(* IEC 61131-3 sources: SafeDODiag/SafeDODiag (part 2) *)

(* ---- DiagAction_InterlockState.st ---- *)
ACTION DiagAction_InterlockState:

	// Check for error state transition and feedback interpretation as long as interlock-based monitoring is enabled
	IF ( Config.InterlockState.EnableMon AND ( Internal.State > SC_INIT ) AND (
		// (Choice 1) if no other monitoring is enabled
		NOT( Config.DiagCode.EnableMon OR Config.Fdbk.EnableMon OR Config.Current.EnableMon ) OR
		// (Choice 2) if DiagCode monitoring is enabled, show Interlock monitoring-based DiagText only when DiagCode indicates "de-energized"
		( Internal.Input.SF_In_DiagCode = 16#8010 )	OR
		// (Choice 3) if any other monitoring is enabled, show Interlock monitoring-based DiagText whenever output is de-energized
		( NOT( Config.DiagCode.EnableMon ) AND ( Config.Fdbk.EnableMon OR Config.Current.EnableMon ) AND NOT( Internal.Input.SO_In_Output1PhysicalState AND Internal.Input.SO_In_Output2PhysicalState ) )
		) ) THEN
		// Go to error state if any error is reported by SO card; the most severe error is prioritized over mixed severities
		IF		Internal.Input.InterlockStateOutput1 = 16#0 // no SafeModuleOK
			OR	Internal.Input.InterlockStateOutput2 = 16#0 // no SafeModuleOK
			THEN
			DiagCode			:= 16#C300;
			Diag.ErrorInterlock	:= TRUE;
			Diag.DiagText		:= 'SafeDOCardOkTimeout';
		ELSIF	Internal.Input.InterlockStateOutput2 = 16#A // hardware/wiring error on output card/channel
			AND	Internal.Input.InterlockStateOutput1 = 16#A // hardware/wiring error on output card/channel
			THEN
			DiagCode			:= 16#C330;
			Diag.ErrorInterlock	:= TRUE;
			Diag.DiagText		:= 'SafeDOCardOutputsHwErr';
		ELSIF	Internal.Input.InterlockStateOutput2 = 16#A // hardware/wiring error on output card/channel
			THEN
			DiagCode			:= 16#C320;
			Diag.ErrorInterlock	:= TRUE;
			Diag.DiagText		:= 'SafeDOCardOutput2HwErr';
		ELSIF	Internal.Input.InterlockStateOutput1 = 16#A // hardware/wiring error on output card/channel
			THEN
			DiagCode			:= 16#C310;
			Diag.ErrorInterlock	:= TRUE;
			Diag.DiagText		:= 'SafeDOCardOutput1HwErr';
			// Except 16#C300, 16#C310, 16#C320, and 16#C330 (above), all else (below) indicate safety CPU programming errors
		ELSIF	Internal.Input.InterlockStateOutput2 = 16#5 // ReleaseOutput and SafeDigitalOutput activate at the same time
			AND	Internal.Input.InterlockStateOutput1 = 16#5 // ReleaseOutput and SafeDigitalOutput activate at the same time
			THEN
			DiagCode			:= 16#C333;
			Diag.ErrorInterlock	:= TRUE;
			Diag.DiagText		:= 'SafeDOCardOutputsSameTimePosEdgePermissionPosEdgeRelease';
		ELSIF	Internal.Input.InterlockStateOutput2 = 16#5 // ReleaseOutput and SafeDigitalOutput activate at the same time
			THEN
			DiagCode			:= 16#C322;
			Diag.ErrorInterlock	:= TRUE;
			Diag.DiagText		:= 'SafeDOCardOutput2SameTimePosEdgePermissionPosEdgeRelease';
		ELSIF	Internal.Input.InterlockStateOutput1 = 16#5 // ReleaseOutput and SafeDigitalOutput activate at the same time
			THEN
			DiagCode			:= 16#C311;
			Diag.ErrorInterlock	:= TRUE;
			Diag.DiagText		:= 'SafeDOCardOutput1SameTimePosEdgePermissionPosEdgeRelease';
		ELSIF	Internal.Input.InterlockStateOutput2 = 16#6 // ReleaseOutput already active when SafeDigitalOutput activates
			AND	Internal.Input.InterlockStateOutput1 = 16#6 // ReleaseOutput already active when SafeDigitalOutput activates
			THEN
			DiagCode			:= 16#C303;
			Diag.ErrorInterlock	:= TRUE;
			Diag.DiagText		:= 'SafeDOCardOutputsPosReleaseBeforePosEdgePermissioin';
		ELSIF	Internal.Input.InterlockStateOutput2 = 16#6 // ReleaseOutput already active when SafeDigitalOutput activates
			THEN
			DiagCode			:= 16#C302;
			Diag.ErrorInterlock	:= TRUE;
			Diag.DiagText		:= 'SafeDOCardOutput2PosReleaseBeforePosEdgePermissioin';
		ELSIF	Internal.Input.InterlockStateOutput1 = 16#6 // ReleaseOutput already active when SafeDigitalOutput activates
			THEN
			DiagCode			:= 16#C301;
			Diag.ErrorInterlock	:= TRUE;
			Diag.DiagText		:= 'SafeDOCardOutput1PosReleaseBeforePosEdgePermissioin';
		ELSIF	( Internal.Input.InterlockStateOutput1 <> 4 AND Internal.Input.InterlockStateOutput1 <> 7 AND Internal.Input.InterlockStateOutput1 <> 8 AND Internal.Input.InterlockStateOutput1 <> 9 )
			OR	( Internal.Input.InterlockStateOutput2 <> 4 AND Internal.Input.InterlockStateOutput2 <> 7 AND Internal.Input.InterlockStateOutput2 <> 8 AND Internal.Input.InterlockStateOutput2 <> 9 )
			THEN
			DiagCode			:= 16#CFFF;
			Diag.ErrorInternal	:= TRUE;
			Diag.DiagText		:= 'UndocumentedError';
		END_IF

		IF ( Diag.ErrorInterlock ) THEN
			Internal.StateGoTo	:= SC_ERROR;
		ELSE
			// both contactor outputs are expected to change interlock states together, so only one channel needs to satisfy the prioritized state check
			IF		( Internal.Input.InterlockStateOutput1 = 16#8 )
				OR	( Internal.Input.InterlockStateOutput2 = 16#8 ) THEN
				DiagCode		:= 16#8100;
				Diag.DiagText	:= 'RequireSafePermission';
			ELSIF	( Internal.Input.InterlockStateOutput1 = 16#7 )
				OR	( Internal.Input.InterlockStateOutput2 = 16#7 ) THEN
				DiagCode		:= 16#8010;
				Diag.DiagText	:= 'RequireOutReq';
			ELSIF	( Internal.Input.InterlockStateOutput1 = 16#4 )
				OR	( Internal.Input.InterlockStateOutput2 = 16#4 ) THEN
				// SO channel is waiting for ReleaseOutput, which should be auto-triggered by safety CPU a few ms after it sets SafeDigitalOutput
				DiagCode		:= 16#8101;
				Diag.DiagText	:= 'RequireSafeRelease';
			END_IF
		END_IF

	END_IF

END_ACTION

(* ---- SimAction_DiagCode.st ---- *)
ACTION SimAction_DiagCode:

	IF ( Simulation.Input.SF_In_DiagCode < 16#C000 ) THEN
		// both outputs are expected to energize together, so either output acting alone will be treated as outputs not energized
		IF ( Simulation.Input.SO_In_Output1PhysicalState AND Simulation.Input.SO_In_Output2PhysicalState ) THEN
			Simulation.Input.SF_In_DiagCode	:= 16#8000;
		ELSE
			Simulation.Input.SF_In_DiagCode	:= 16#8010;
		END_IF
		// simulate SF_EDM response after monitor time is over
		Internal.Fub.TON_EDMMonitorSim.IN := ( Simulation.Input.SO_In_Output1PhysicalState = Internal.Prev.SimOutput1 ) AND ( Simulation.Input.SO_In_Output2PhysicalState = Internal.Prev.SimOutput2 );
		IF ( Internal.Fub.TON_EDMMonitorSim.IN AND Internal.Fub.TON_EDMMonitorSim.Q ) THEN
			// both outputs are expected to energize together, so either output acting alone will be treated as outputs not energized
			IF ( NOT ( Simulation.Input.SO_In_Output1PhysicalState AND Simulation.Input.SO_In_Output2PhysicalState ) AND Simulation.Input.SI_In_Contactor1Fdbk AND Simulation.Input.SI_In_Contactor2Fdbk ) THEN
				Simulation.Input.SF_In_DiagCode	:= 16#8010;
			ELSIF ( NOT ( Simulation.Input.SO_In_Output1PhysicalState AND Simulation.Input.SO_In_Output2PhysicalState ) AND NOT Simulation.Input.SI_In_Contactor1Fdbk AND Simulation.Input.SI_In_Contactor2Fdbk ) THEN
				Simulation.Input.SF_In_DiagCode	:= 16#C040;
			ELSIF ( NOT ( Simulation.Input.SO_In_Output1PhysicalState AND Simulation.Input.SO_In_Output2PhysicalState ) AND Simulation.Input.SI_In_Contactor1Fdbk AND NOT Simulation.Input.SI_In_Contactor2Fdbk ) THEN
				Simulation.Input.SF_In_DiagCode	:= 16#C050;
			ELSIF ( NOT ( Simulation.Input.SO_In_Output1PhysicalState AND Simulation.Input.SO_In_Output2PhysicalState ) AND NOT Simulation.Input.SI_In_Contactor1Fdbk AND NOT Simulation.Input.SI_In_Contactor2Fdbk ) THEN
				Simulation.Input.SF_In_DiagCode	:= 16#C060;
			ELSIF ( Simulation.Input.SO_In_Output1PhysicalState AND Simulation.Input.SO_In_Output2PhysicalState AND Simulation.Input.SI_In_Contactor1Fdbk AND Simulation.Input.SI_In_Contactor2Fdbk ) THEN
				Simulation.Input.SF_In_DiagCode	:= 16#C090;
			ELSIF ( Simulation.Input.SO_In_Output1PhysicalState AND Simulation.Input.SO_In_Output2PhysicalState AND NOT Simulation.Input.SI_In_Contactor1Fdbk AND Simulation.Input.SI_In_Contactor2Fdbk ) THEN
				Simulation.Input.SF_In_DiagCode	:= 16#C080;
			ELSIF ( Simulation.Input.SO_In_Output1PhysicalState AND Simulation.Input.SO_In_Output2PhysicalState AND Simulation.Input.SI_In_Contactor1Fdbk AND NOT Simulation.Input.SI_In_Contactor2Fdbk ) THEN
				Simulation.Input.SF_In_DiagCode	:= 16#C070;
			ELSIF ( Simulation.Input.SO_In_Output1PhysicalState AND Simulation.Input.SO_In_Output2PhysicalState AND NOT Simulation.Input.SI_In_Contactor1Fdbk AND NOT Simulation.Input.SI_In_Contactor2Fdbk ) THEN
				Simulation.Input.SF_In_DiagCode	:= 16#8000;
			END_IF
			// check for static TRUE signal on EDM reset at the time error occurs
			IF ( Status.SafetyResetRequested AND Simulation.Input.SF_In_DiagCode >= 16#C000 ) THEN
				Simulation.Input.SF_In_DiagCode	:= Simulation.Input.SF_In_DiagCode + 1;
			END_IF
		END_IF
	ELSE
		Internal.Fub.TON_EDMMonitorSim.IN := FALSE;
		IF ( Status.SafetyResetRequested ) THEN
			Simulation.Input.SF_In_DiagCode	:= 16#8010;
		END_IF
	END_IF

END_ACTION

(* ---- StateAction_CommonAft.st ---- *)
ACTION StateAction_CommmonAft:

	// Run timers
	Internal.Fub.TON_EDMMonitorSim.PT	:= T#200ms;
	Internal.Fub.TON_EDMMonitorSim();
	Internal.Fub.TON_EDMStartDelay.PT	:= Config.DiagCode.StartDelayTime;
	Internal.Fub.TON_EDMStartDelay();
	Internal.Fub.TON_EDMResetDelay.PT	:= Config.DiagCode.ResetDelayTime;
	Internal.Fub.TON_EDMResetDelay();
	Internal.Fub.TON_FdbkStartDelay.PT	:= Config.Fdbk.StartDelayTime;
	Internal.Fub.TON_FdbkStartDelay();
	Internal.Fub.TON_Fdbk.PT			:= Config.Fdbk.MonitorTime;
	Internal.Fub.TON_Fdbk();
	Internal.Fub.TON_Current.PT			:= Config.Current.MonitorTime;
	Internal.Fub.TON_Current();
	Internal.Fub.TON_InterlockStartDelay.PT	:= Config.InterlockState.StartDelayTime;
	Internal.Fub.TON_InterlockStartDelay();
	Internal.Fub.TON_Interlock.PT			:= Config.InterlockState.MonitorTime;
	Internal.Fub.TON_Interlock();
	// Reset timers by default and wait for the state machine to override the default, so any state transition that's
	// not made within the state machine (e.g. global jump into error state) will automatically disable abandoned timers
	Internal.Fub.TON_EDMStartDelay.IN		:= FALSE;
	Internal.Fub.TON_FdbkStartDelay.IN		:= FALSE;
	Internal.Fub.TON_Fdbk.IN				:= FALSE;
	Internal.Fub.TON_Current.IN				:= FALSE;
	Internal.Fub.TON_InterlockStartDelay.IN	:= FALSE;
	Internal.Fub.TON_Interlock.IN			:= FALSE;
	IF ( Internal.State <> SC_ERROR ) THEN
		Internal.Fub.TON_EDMResetDelay.IN	:= FALSE;
	END_IF

	// Help to check for changes in input values
	Internal.Prev.Reset			:= Cmd.Reset;
	Internal.Prev.EnDiagCode	:= Config.DiagCode.EnableMon;
	Internal.Prev.EnFdbk		:= Config.Fdbk.EnableMon;
	Internal.Prev.EnCurrent		:= Config.Current.EnableMon;
	Internal.Prev.EnInterlock	:= Config.InterlockState.EnableMon;
	Internal.Prev.SimOutput1	:= Simulation.Input.SO_In_Output1PhysicalState;
	Internal.Prev.SimOutput2	:= Simulation.Input.SO_In_Output2PhysicalState;

END_ACTION

(* ---- StateAction_CommonPre.st ---- *)
ACTION StateAction_CommonPre:

	//########## Feedback interpretation and error state transition ##########
	// Check for error state transition that apply no matter what state the fub was in
	IF ( Error ) THEN
		// Go to error state if a process error was detected (e.g. fub cfg error, 2-channel switching discrepancy, undocumented error code)
		Internal.StateGoTo	:= SC_ERROR;

	ELSIF	( Config.DiagCode.EnableMon AND NOT( Internal.Prev.EnDiagCode ) )
		OR	( Config.Fdbk.EnableMon AND NOT( Internal.Prev.EnFdbk ) )
		OR	( Config.Current.EnableMon AND NOT( Internal.Prev.EnCurrent ) )
		OR	( Config.InterlockState.EnableMon AND NOT( Internal.Prev.EnInterlock ) ) THEN
		Internal.StateGoTo	:= SC_CFG;
		Diag.DiagText		:= '';
		DiagCode			:= 0;

		// Exclusively for DiagCode-based monitoring:
	ELSIF ( Config.DiagCode.EnableMon AND ( Internal.State > SC_INIT OR Internal.State = SC_ERROR ) ) THEN
		DiagAction_DiagCode;
	END_IF

	// Check for error state transition and feedback interpretation as long as interlock-based monitoring is enabled
	DiagAction_InterlockState;

	// Keep track of state changes
	Internal.Prev.State	:= Internal.State;
	Internal.State		:= Internal.StateGoTo;

END_ACTION

(* ---- StateAction_Disabled.st ---- *)
ACTION StateAction_Disabled:

	//#################### Check the SF_EDM fub DiagCode ##################
	// if DiagCode is checked, error flagged at the beginning of the fub will put the state machine into error state and skip this state
	// while non-zero DiagCode would update the DiagText at the beginning of the fub
	IF ( Config.DiagCode.EnableMon ) THEN

		CASE Internal.Input.SF_In_DiagCode OF
			16#0000:
			DiagCode		:= 16#0003;
			Diag.DiagText	:= 'WaitingForSafeFubComm';
			16#8000:
			Internal.StateGoTo	:= SC_ENABLED;
		END_CASE

	//#################### Check the contactor feedback ##################
	ELSIF ( Config.Fdbk.EnableMon ) THEN

		// both fdbks need to be active (to show that both contactors are open); if either fdbk is inactive, start the fdbk timer to check if they activate before timeout
		Internal.Fub.TON_Fdbk.IN := NOT( Internal.Input.SI_In_Contactor1Fdbk AND Internal.Input.SI_In_Contactor2Fdbk );

		// Go to enabled state if SO card outputs are physically active during operation
		IF ( Internal.Input.SO_In_Output1PhysicalState AND Internal.Input.SO_In_Output2PhysicalState ) THEN
			Internal.Fub.TON_Fdbk.IN := FALSE;

			Internal.StateGoTo	:= SC_ENABLED;
			DiagCode			:= 16#8000;
			Diag.DiagText		:= 'Energized';

		ELSIF ( Internal.Fub.TON_Fdbk.Q ) THEN
			Internal.Fub.TON_Fdbk.IN := FALSE;
			Diag.ErrorFdbk := TRUE; // set the error flag and it will put the state machine into error state

			IF ( Internal.Input.SI_In_Contactor1Fdbk ) THEN
				DiagCode		:= 16#C050;
				Diag.DiagText	:= 'NegFdbk2AfterNegOutReq';
			ELSIF ( Internal.Input.SI_In_Contactor2Fdbk ) THEN
				DiagCode		:= 16#C040;
				Diag.DiagText	:= 'NegFdbk1AfterNegOutReq';
			ELSE
				DiagCode		:= 16#C060;
				Diag.DiagText	:= 'NegFdbkAfterNegOutReq';
			END_IF

		ELSIF NOT( Config.InterlockState.EnableMon ) THEN
			DiagCode			:= 16#8110;
			Diag.DiagText		:= 'De-energized';
		END_IF

	//#################### Check the output current ##################
	ELSIF ( Config.Current.EnableMon ) THEN

		// if either SO card output current is maintained or if contactor current is above threshold, start the current timer to check if they deactivate before timeout
		Internal.Fub.TON_Current.IN := Internal.Input.SO_In_Output1CurrentOK OR Internal.Input.SO_In_Output2CurrentOK;

		// Go to enabled state if SO card outputs are physically active during operation
		IF ( Internal.Input.SO_In_Output1PhysicalState AND Internal.Input.SO_In_Output2PhysicalState ) THEN
			Internal.Fub.TON_Current.IN := FALSE;

			Internal.StateGoTo	:= SC_ENABLED;
			DiagCode			:= 16#8000;
			Diag.DiagText		:= 'Energized';

		ELSIF ( Internal.Fub.TON_Current.Q) THEN
			Internal.Fub.TON_Current.IN	:= FALSE;
			Diag.ErrorCurrent := TRUE; // set the error flag and it will put the state machine into error state

			IF NOT( Internal.Input.SO_In_Output1CurrentOK ) THEN
				DiagCode		:= 16#C250;
				Diag.DiagText	:= 'PosCurrentOk2AfterNegOutReq';
			ELSIF NOT( Internal.Input.SO_In_Output2CurrentOK ) THEN
				DiagCode		:= 16#C240;
				Diag.DiagText	:= 'PosCurrentOk1fterNegOutReq';
			ELSE
				DiagCode		:= 16#C260;
				Diag.DiagText	:= 'PosCurrentOkAfterNegOutReq';
			END_IF

		ELSIF NOT( Config.InterlockState.EnableMon ) THEN
			DiagCode			:= 16#8110;
			Diag.DiagText		:= 'De-energized';
		END_IF

	//#################### Check the output interlock ##################
	// if interlock state is checked, error flagged at the beginning of the fub will put the state machine into error state and skip this state
	ELSIF ( Config.InterlockState.EnableMon ) THEN

		IF	Internal.Input.InterlockStateOutput2 = 16#9 // output energized
			AND	Internal.Input.InterlockStateOutput1 = 16#9 // output energized
			THEN
			Internal.StateGoTo	:= SC_ENABLED;
			DiagCode			:= 16#8000;
			Diag.DiagText		:= 'Energized';
		ELSE
			// if only one output is enabled, start the interlock timer to check if the other output enables before timeout
			Internal.Fub.TON_Interlock.IN := ( Internal.Input.InterlockStateOutput1 = 16#9 ) XOR ( Internal.Input.InterlockStateOutput2 = 16#9 );

			IF ( Internal.Fub.TON_Interlock.Q ) THEN
				Internal.Fub.TON_Interlock.IN := FALSE;
				Diag.ErrorInterlock	:= TRUE; // set the error flag and it will put the state machine into error state
				DiagCode			:= 16#C340;
				Diag.DiagText		:= 'SafeDOCardPosOutputsNotSameTime';
			END_IF
		END_IF

	//#################### Show state text and check transitions when there is no monitoring ####################
	ELSE
		// Go to enabled state if SO card outputs are physically active during operation
		IF ( Internal.Input.SO_In_Output1PhysicalState AND Internal.Input.SO_In_Output2PhysicalState ) THEN
			Internal.StateGoTo	:= SC_ENABLED;
			DiagCode			:= 16#8000;
			Diag.DiagText		:= 'Energized';
		ELSE
			DiagCode			:= 16#8110;
			Diag.DiagText		:= 'De-energized';
		END_IF
	END_IF

END_ACTION

(* ---- StateAction_Enabled.st ---- *)
ACTION StateAction_Enabled:

	//#################### Check the SF_EDM fub DiagCode ##################
	// if DiagCode is checked, error flagged at the beginning of the fub will put the state machine into error state and skip this state
	// while non-zero DiagCode would update the DiagText at the beginning of the fub
	IF ( Config.DiagCode.EnableMon ) THEN

		IF ( Internal.Input.SF_In_DiagCode <> 16#8000 ) THEN
			Internal.StateGoTo	:= SC_DISABLED;
		END_IF

	//#################### Check the contactor feedback ##################
	ELSIF ( Config.Fdbk.EnableMon ) THEN

		// both fdbks need to be inactive (to mean that both contactors are closed); if either fdbk is active, start the fdbk timer to check if they deactivate before timeout
		Internal.Fub.TON_Fdbk.IN := ( Internal.Input.SI_In_Contactor1Fdbk OR Internal.Input.SI_In_Contactor2Fdbk );

		// Go to disabled state if SO card outputs are not both physically active during operation
		IF ( NOT( Internal.Input.SO_In_Output1PhysicalState AND Internal.Input.SO_In_Output2PhysicalState ) ) THEN
			Internal.Fub.TON_Current.IN := FALSE;

			Internal.StateGoTo	:= SC_DISABLED;
			IF NOT( Config.InterlockState.EnableMon ) THEN
				DiagCode		:= 16#8110;
				Diag.DiagText	:= 'De-energized';
			END_IF

		ELSIF ( Internal.Fub.TON_Fdbk.Q ) THEN
			Internal.Fub.TON_Fdbk.IN := FALSE;
			Diag.ErrorFdbk := TRUE; // set the error flag and it will put the state machine into error state

			IF NOT( Internal.Input.SI_In_Contactor1Fdbk ) THEN
				DiagCode		:= 16#C080;
				Diag.DiagText	:= 'PosFdbk2AfterPosOutReq';
			ELSIF NOT( Internal.Input.SI_In_Contactor2Fdbk ) THEN
				DiagCode		:= 16#C070;
				Diag.DiagText	:= 'PosFdbk1AfterPosOutReq';
			ELSE
				DiagCode		:= 16#C090;
				Diag.DiagText	:= 'PosFdbkAfterPosOutReq';
			END_IF

		ELSE
			DiagCode			:= 16#8000;
			Diag.DiagText		:= 'Energized';
		END_IF

	//#################### Check the output current ##################
	ELSIF ( Config.Current.EnableMon ) THEN

		// if both SO card output currents are not okay or if contactor current isn't above threshold, start the current timer to check if they normalize before timeout
		Internal.Fub.TON_Current.IN := NOT( Internal.Input.SO_In_Output1CurrentOK AND Internal.Input.SO_In_Output2CurrentOK );

		// Go to disabled state if SO card outputs are not both physically active during operation
		IF ( NOT( Internal.Input.SO_In_Output1PhysicalState AND Internal.Input.SO_In_Output2PhysicalState ) ) THEN
			Internal.Fub.TON_Current.IN := FALSE;

			Internal.StateGoTo	:= SC_DISABLED;
			IF NOT( Config.InterlockState.EnableMon ) THEN
				DiagCode		:= 16#8110;
				Diag.DiagText	:= 'De-energized';
			END_IF

		ELSIF ( Internal.Fub.TON_Current.Q) THEN
			Internal.Fub.TON_Current.IN := FALSE;
			Diag.ErrorCurrent := TRUE; // set the error flag and it will put the state machine into error state

			IF ( Internal.Input.SO_In_Output1CurrentOK ) THEN
				DiagCode		:= 16#C280;
				Diag.DiagText	:= 'NegCurrentOk2AfterPosOutReq';
			ELSIF ( Internal.Input.SO_In_Output2CurrentOK ) THEN
				DiagCode		:= 16#C270;
				Diag.DiagText	:= 'NegCurrentOk1AfterPosOutReq';
			ELSE
				DiagCode		:= 16#C290;
				Diag.DiagText	:= 'NegCurrentOkAfterPosOutReq';
			END_IF

		ELSE
			DiagCode			:= 16#8000;
			Diag.DiagText		:= 'Energized';
		END_IF

	//#################### Check the output interlock ##################
	ELSIF ( Config.InterlockState.EnableMon ) THEN
		// if interlock state is checked, error flagged at the beginning of the fub will put the state machine into error state and skip this state
		IF NOT( Internal.Input.InterlockStateOutput2 = 16#9
			AND	Internal.Input.InterlockStateOutput1 = 16#9 )
			THEN // one or both outputs not energized
			Internal.StateGoTo	:= SC_DISABLED;
		END_IF

	ELSE
		//#################### Show state text and check transitions when there is no monitoring ####################
		// Stay in enabled state if SO card outputs are physically active during operation
		IF ( ( Internal.Input.SO_In_Output1PhysicalState AND Internal.Input.SO_In_Output2PhysicalState ) ) THEN
			DiagCode			:= 16#8000;
			Diag.DiagText		:= 'Energized';
		ELSE
			Internal.StateGoTo	:= SC_DISABLED;
			DiagCode			:= 16#8110;
			Diag.DiagText		:= 'De-energized';
		END_IF
	END_IF

END_ACTION

(* ---- StateAction_Error.st ---- *)
ACTION StateAction_Error:

	// Only clear fub error on the rising edge of reset request
			// Reset Error and DiagCode outputs if alarms were acknowledged by command or via reset in the alarm system
	IF( Cmd.Reset AND NOT( Internal.Prev.Reset ) )THEN
		IF ( Diag.ErrorConfig ) THEN
			Diag.ErrorConfig	:= FALSE;
			Diag.DiagText		:= '';
			DiagCode			:= 0;
			// Go back to the config state
			Internal.StateGoTo	:= SC_CFG;
		ELSIF ( Diag.ErrorSafeFub ) THEN
			// Give SF_EDM fub enough time to react to error reset
			Internal.Fub.TON_EDMResetDelay.IN := TRUE;
			Internal.EDMReset	:= TRUE;
		ELSE
			Diag.ErrorFdbk		:= FALSE;
			Diag.ErrorCurrent	:= FALSE;
			Diag.ErrorInterlock	:= FALSE;
			Diag.DiagText		:= '';
			DiagCode			:= 0;
			// Go into the disabled state
			Internal.StateGoTo	:= SC_DISABLED;
		END_IF
	END_IF

	// After EDM reset delay timeout, go into the disabled state
	IF ( Internal.Fub.TON_EDMResetDelay.Q ) THEN
		Internal.Fub.TON_EDMResetDelay.IN := FALSE;
		Diag.ErrorSafeFub	:= FALSE;
		Diag.DiagText		:= '';
		DiagCode			:= 0;
		Internal.EDMReset	:= FALSE;
		Internal.StateGoTo	:= SC_DISABLED;
	END_IF

END_ACTION

(* ---- StateAction_Init.st ---- *)
ACTION StateAction_Init:

	//#################### Check startup timing error of SF_EDM fub DiagCode monitor ##################
	IF Config.DiagCode.EnableMon THEN
		DiagCode := Internal.Input.SF_In_DiagCode;
		// If SF_EDM DiagCode monitoring is enabled, start the delay timer to give safety CPU's SF_EDM fub enough time (>= MonitorTime) to report that contactors are not open (DiagCode 16#C060)
		Internal.Fub.TON_EDMStartDelay.IN := Internal.Input.SI_In_SafeModuleOK;

		IF ( Internal.Fub.TON_EDMStartDelay.Q ) THEN
			Internal.Fub.TON_EDMStartDelay.IN := FALSE;

			// Already waited for SF_EDM fub to report stabilized DiagCode but got no response
			IF ( Internal.Input.SF_In_DiagCode = 0 ) THEN
				DiagCode			:= 16#C000;
				Diag.ErrorSafeFub	:= TRUE;
				Diag.DiagText		:= 'SafeFubCommTimeout';

				// Check if safety application is operational and SF_EDM reports no error
			ELSIF ( Internal.Input.SF_In_DiagCode < 16#C000 ) THEN
				DiagCode			:= Internal.Input.SF_In_DiagCode;
				IF ( Internal.Input.SF_In_DiagCode = 16#8000 ) THEN
					Internal.StateGoTo	:= SC_ENABLED;
				ELSE
					Internal.StateGoTo	:= SC_DISABLED;
				END_IF

				// Check if a start reset of safety CPU's SF_EDM fub is necessary (for situations where the gray CPU reboots but the safety CPU isn't power cycled)
			ELSIF ( Internal.Input.SF_In_DiagCode = 16#C060 ) THEN
				// Start the reset delay timer to give SF_EDM fub enough time to report that contactors are indeed open:
				// Following fdbk SI card's SafeModuleOK, safety CPU may need extra time to determine SI card channels are OK
				Internal.Fub.TON_EDMResetDelay.IN := TRUE;

				// if contactors show to be open (feedbacks are TRUE) before timeout, request a safety reset
				IF ( Internal.Input.SI_In_Contactor1Fdbk AND Internal.Input.SI_In_Contactor2Fdbk AND NOT( Internal.EDMReset ) ) THEN
					//Internal.Fub.TON_EDMResetDelay.IN	:= FALSE; //--> the timer shouldn't need to restart because safety CPU's reaction to the reset request should be included in the timer preset
					Internal.EDMReset	:= TRUE;
					DiagCode			:= 16#8001;
					Diag.DiagText		:= 'RequireStartReset';
					// if timeout happens (e.g. actual feedback error or gray CPU doesn't send SF_EDM reset request to safety CPU), set the error flag and it will put the state machine into error state
				ELSIF ( Internal.Fub.TON_EDMResetDelay.Q ) THEN
					Internal.Fub.TON_EDMResetDelay.IN := FALSE;
					Internal.EDMReset	:= FALSE;
					DiagCode			:= Internal.Input.SF_In_DiagCode;
					Diag.ErrorSafeFub	:= TRUE;
				END_IF

				// For all other DiagCodes, set the error flag and it will put the state machine into error state
			ELSE
				DiagCode			:= Internal.Input.SF_In_DiagCode;
				Diag.ErrorSafeFub	:= TRUE;

			END_IF

		ELSE
			IF ( Internal.Input.SI_In_SafeModuleOK ) THEN
				// Wait for SF_EDM fub to report stabilized DiagCode because it is likely to report 16#8010 until MonitorTime has passed
				DiagCode		:= 16#0003;
				Diag.DiagText	:= 'WaitingForSafeFubComm';
			ELSE
				DiagCode		:= 16#0002;
				Diag.DiagText	:= 'WaitingForSafeDIComm';
			END_IF
		END_IF // end DiagCode start delay

		//#################### Check startup timing error of Contactor Feedback monitor ####################
	ELSIF Config.Fdbk.EnableMon THEN
		// If feedback monitoring is enabled, start the delay timer to give fdbk SI card enough time to report that contactors are indeed open:
		// Following fdbk SI card's SafeModuleOK, safety CPU may need extra time to determine SI card channels are OK
		Internal.Fub.TON_FdbkStartDelay.IN := Internal.Input.SI_In_SafeModuleOK;

		// Check if contactors show to be open (feedbacks are TRUE) before timeout
		IF ( Internal.Input.SI_In_Contactor1Fdbk AND Internal.Input.SI_In_Contactor2Fdbk AND NOT( Internal.EDMReset ) ) THEN
			//Internal.Fub.TON_FdbkStartDelay.IN := FALSE; //--> the timer shouldn't need to restart because safety CPU's reaction to the reset request should be included in the timer preset
			Internal.EDMReset	:= TRUE;
			DiagCode			:= 16#8002;
			Diag.DiagText		:= 'MayRequireStartReset';

		ELSIF ( Internal.Fub.TON_FdbkStartDelay.Q ) THEN
			Internal.Fub.TON_FdbkStartDelay.IN := FALSE;
			Internal.EDMReset	:= FALSE;

			// if contactors are open when timeout happens, assume SF_EDM fub error has cleared
			IF ( Internal.Input.SI_In_Contactor1Fdbk AND Internal.Input.SI_In_Contactor2Fdbk ) THEN
				Internal.StateGoTo	:= SC_DISABLED;
				DiagCode			:= 16#8110;
				Diag.DiagText		:= 'De-energized';
				// if contactor 2 is open when timeout happens, set the fdbk 1 error flag and it will put the state machine into error state
			ELSIF ( Internal.Input.SI_In_Contactor2Fdbk ) THEN
				DiagCode		:= 16#C040;
				Diag.ErrorFdbk	:= TRUE;
				Diag.DiagText	:= 'NegFdbk1AfterNegOutReq';
				// if contactor 1 is open when timeout happens, set the fdbk 2 error flag and it will put the state machine into error state
			ELSIF ( Internal.Input.SI_In_Contactor1Fdbk ) THEN
				DiagCode		:= 16#C050;
				Diag.ErrorFdbk	:= TRUE;
				Diag.DiagText	:= 'NegFdbk2AfterNegOutReq';
				// if both contactors are closed when timeout happens, set the error flag and it will put the state machine into error state
			ELSE
				DiagCode		:= 16#C060;
				Diag.ErrorFdbk	:= TRUE;
				Diag.DiagText	:= 'NegFdbk1Fdbk2AfterNegOutReq';
			END_IF

		ELSE
			DiagCode		:= 16#0002;
			Diag.DiagText	:= 'WaitingForSafeDIComm';
		END_IF // end feedback start delay

		//#################### Check startup timing error of Output Interlock monitor ####################
	ELSIF Config.InterlockState.EnableMon THEN
		// If output interlock monitoring is enabled, start the delay timer to give SO card enough time to report that channels are ready:
		// Following SO card's SafeModuleOK, safety CPU may need extra time to determine SO card channels are OK
		Internal.Fub.TON_InterlockStartDelay.IN := Internal.Input.SO_In_SafeModuleOK;

		// Check if output interlock states are ready before timeout
		IF ( Internal.Input.InterlockStateOutput1 > 0 AND Internal.Input.InterlockStateOutput2 > 0 ) THEN
			Internal.Fub.TON_InterlockStartDelay.IN := FALSE;

			Internal.StateGoTo	:= SC_DISABLED;

			// if timeout happens, set the error flag and it will put the state machine into error state
		ELSIF ( Internal.Fub.TON_InterlockStartDelay.Q ) THEN
			Internal.Fub.TON_InterlockStartDelay.IN := FALSE;

			DiagCode			:= 16#C300;
			Diag.ErrorInterlock	:= TRUE;
			Diag.DiagText		:= 'SafeDOCardOkTimeout';

		ELSE
			DiagCode		:= 16#0001;
			Diag.DiagText	:= 'WaitingForSafeDOComm';
		END_IF // end interlock state start delay

		//#################### Ignore startup reset if only current OK monitor is used or if no monitor is used ####################
	ELSE
		// Wait for SO card comm with safety CPU
		IF ( Internal.Input.SO_In_SafeModuleOK ) THEN
			Internal.StateGoTo	:= SC_DISABLED;
			DiagCode			:= 16#8110;
			Diag.DiagText		:= 'De-energized';
		ELSE
			DiagCode		:= 16#0001;
			Diag.DiagText	:= 'WaitingForSafeDOComm';
		END_IF
	END_IF

END_ACTION
